PROGRAM simIniciaProg_Manual
VAR
	bSimIniciaProg: BOOL:= FALSE;
	posicaoAtual: STRING;
	envialog: STRING;
	bGravarConfigPosicao_Reator: BOOL;
END_VAR


gvl_p.arrStatusEstufas[gvl.actEst].startManual := TRUE;

bGravarConfigPosicao_Reator:= TRUE;

END_PROGRAM

(* stored: Version 1.1.0.1, ProductVersion 3.1.4024.12
   POU simIniciaProg_Manual: Id {49aef258-0369-4c54-af1f-b24b3eb016eb}, SpecialFunc None *)
